// TIA Portal V20 export
// export: Created 2025-12-01T14:57:11.7260089Z, ExportSetting None, DisplayName Totally Integrated Automation Portal, DisplayVersion V20 Update 3, DisplayName TIA Portal Openness, DisplayVersion V20 Update 3, DisplayName TIA Portal Version Control Interface, DisplayVersion V20 Update 3, DisplayName STEP 7 Professional, DisplayVersion V20 Update 3, DisplayName STEP 7 Safety, DisplayVersion V20 Update 2, DisplayName WinCC Basic/Comfort/Advanced, DisplayVersion V20 Update 3, DisplayName WinCC Professional, DisplayVersion V20 Update 3, DisplayName WinCC Unified, DisplayVersion V20 Update 3
FUNCTION "FC863_PrimeraUT_EnMesa" : Void   // FC863, STL
{ S7_Optimized_Access := 'FALSE' }
// stored: AutoNumber false
   VAR_INPUT
      Mesa : UInt;
   END_VAR
   VAR_OUTPUT
      PrimeraUT : UInt;
   END_VAR
   VAR_TEMP
      Relleno : Byte;
      ValorReturn : Int;
   END_VAR
BEGIN

NETWORK
TITLE = Inicializar
//////////////////////////////////////////////////////////////////////
/// Inicializar Variables




NETWORK
TITLE = Buscar Primera UT de la Mesa
//////////////////////////////////////////////////////////////////////
/// Buscar Primera UT de la Mesa
      L     "DB810_ColasMesas".Colas[#Mesa].UT_PrimeraMesa;
      T     #PrimeraUT;

      BE;  // - Finalizar bloque


END_FUNCTION
